{attribute 'qualified_only'}
{attribute 'strict'}
TYPE E_LoadPriority :
(
	None := 0,// 无等级
	Line0,// 优先0
	Line1// 优先1
);
END_TYPE

(* stored: Version 1.1.0.1, ProductVersion 3.1.4024.3
   DUT E_LoadPriority: Id {4c3b15bf-9552-4df7-aa75-0dc987267f66} *)
